KUKA KRL data list: FlowControl.dat

&ACCESS RVP
DEFDAT FlowControl Public

DECL CHAR MSG
DECL CHAR STATE
DECL BOOL AVAILABLE

ENDDAT
